(* CODESYS project Esteira SET e RESET .project

Project tree, tasks and I/O mapping:
  Device : CODESYS Control Win V3, 3S - Smart Software Solutions GmbH, order no. 305021, version 3.5.11.30
    application Application
      libraries: Standard, * (System)
      task MainTask (cyclic, interval t#20ms, priority 1) calls PLC_PRG
      program PLC_PRG [LD]
      Symbols
*)

// Device/Application/PLC_PRG
PROGRAM PLC_PRG
VAR
	Start:BOOL; 
	Stop:BOOL;
	Emergencia:BOOL;
	Start_Light:BOOL;
	Stop_Light:BOOL;
	SensorA:BOOL;
	SensorB:BOOL;
	Esteira1:BOOL; 
	Esteira2:BOOL; 
	
	F_TRIG_0: F_TRIG;
END_VAR
VAR // added by the converter: edge detectors and wires of the graphical bodies
    _w1, _w2 : BOOL;
END_VAR

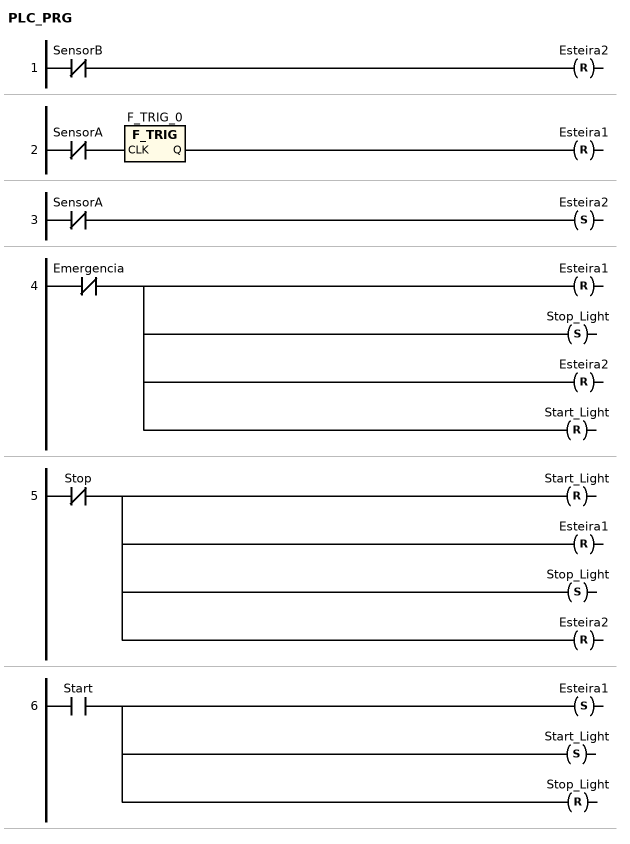
// NETWORK 1
Esteira2 R= NOT SensorB;

// NETWORK 2
F_TRIG_0(CLK := NOT SensorA); // F_TRIG
Esteira1 R= F_TRIG_0.Q;

// NETWORK 3
Esteira2 S= NOT SensorA;

// NETWORK 4
_w1 := NOT Emergencia;
Esteira1 R= _w1;
Stop_Light S= _w1;
Esteira2 R= _w1;
Start_Light R= _w1;

// NETWORK 5
_w2 := NOT Stop;
Start_Light R= _w2;
Esteira1 R= _w2;
Stop_Light S= _w2;
Esteira2 R= _w2;

// NETWORK 6
Esteira1 S= Start;
Start_Light S= Start;
Stop_Light R= Start;

END_PROGRAM
